FUNCTION_BLOCK FB_TestFunctionBlock
VAR
	nCounter : LINT;
END_VAR

nCounter := nCounter + 1;

END_FUNCTION_BLOCK

(* stored: Version 1.1.0.1, ProductVersion 3.1.4024.12
   POU FB_TestFunctionBlock: Id {d572f337-29d2-46df-a865-e75df6da31ee}, SpecialFunc None *)
